FUNCTION_BLOCK FieldsToServiceRequestForm (* Translate individual fields to a ServiceRequestForm type *)
  (* Standard: 61499-2; Description: Copyright (c) 2018 fortiss GmbH This program and the accompanying materials are made available under the terms of the Eclipse Public License 2.0 which is available at https://www.eclipse.org/legal/epl-2.0/ SPDX-License-Identifier: EPL-2.0 *)
  (* Version 1.0, 2018-08-21, Jose Cabral, fortiss GmbH *)
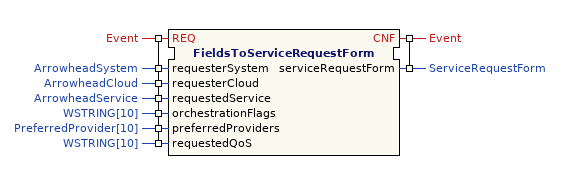
  EVENT_INPUT
    REQ WITH requesterSystem, requesterCloud, requestedQoS, preferredProviders, orchestrationFlags, requestedService; (* Create ServiceRequestForm *)
  END_EVENT
  EVENT_OUTPUT
    CNF WITH serviceRequestForm; (* ServiceRequestForm  created *)
  END_EVENT
  VAR_INPUT
    requesterSystem : ArrowheadSystem; (* The ArrowheadSystem identifier that is requesting the orchestration *)
    requesterCloud : ArrowheadCloud; (* Not to be used by Application Systems. This field is only used when there is an inbound request from another Cloud. This can only be submitted by the Gatekeeper *)
    requestedService : ArrowheadService; (* When not filled out, the Orchestrator operate in the ”default configuration” mode. When filled out, other fields will affect how the orchestration will work – but the Service will be specified by the Consumer in advance then *)
    orchestrationFlags : ARRAY [0..9] OF WSTRING; (* These flags can be set to tailor the orchestration process (use just the names of the flags to be enabled) *)
    preferredProviders : ARRAY [0..9] OF PreferredProvider; (* There can be a list from the Consumer stating which other Application Systems (even from other Clouds) it wishes to connect. If this field is filled out, the Orchestrator will try to facilitate these preferences *)
    requestedQoS : ARRAY [0..9] OF WSTRING; (* This object will be presenting the Consumer’s selected QoS level. Not implemented *)
  END_VAR
  VAR_OUTPUT
    serviceRequestForm : ServiceRequestForm; (* Created ServiceRequestForm *)
  END_VAR
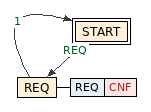
  EC_STATES
    START; (* Initial State *)
    REQ : REQ -> CNF; (* Normal execution *)
  END_STATES
  EC_TRANSITIONS
    START TO REQ := REQ;
    REQ TO START := 1;
  END_TRANSITIONS
  ALGORITHM REQ IN ST: (* Normally executed algorithm *)
VAR
  i: INT;
END_VAR;

serviceRequestForm.requesterSystem := requesterSystem;
serviceRequestForm.requesterCloud := requesterCloud;
serviceRequestForm.requestedService := requestedService;


i := 0;
WHILE i < 10 DO //looks like while is faster than FOR when exporting to cpp
  serviceRequestForm.orchestrationFlags[i] :=  orchestrationFlags[i];
  serviceRequestForm.preferredProviders[i] := preferredProviders[i];
  serviceRequestForm.requestedQoS[i] := requestedQoS[i];
  i := i + 1;
END_WHILE
  END_ALGORITHM
END_FUNCTION_BLOCK
